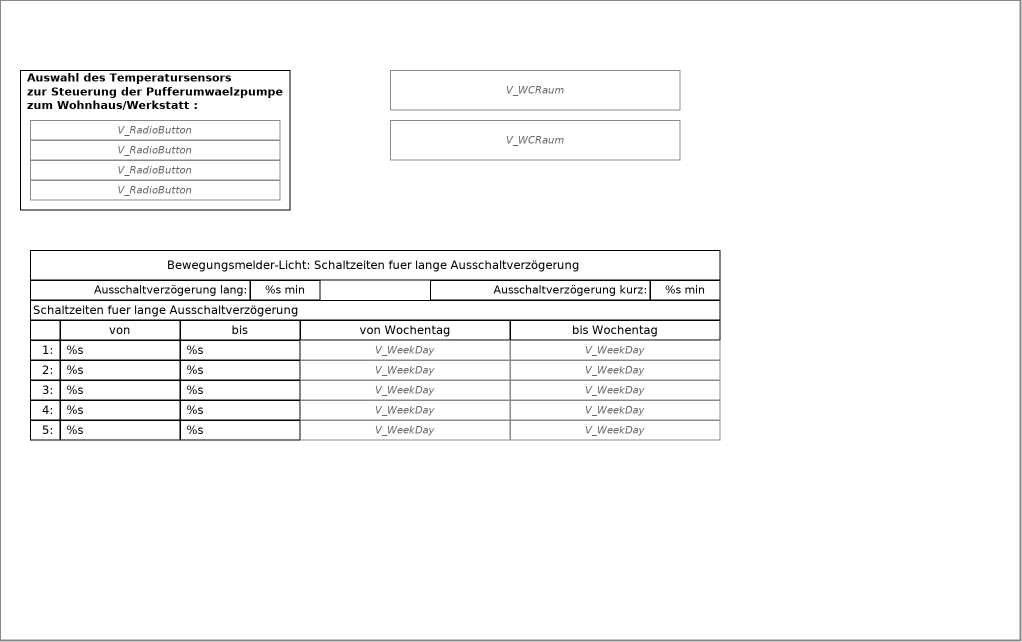
VISUALIZATION V_Einstellungen  // 1022x642
    Frame (0,-120 1020x760)
        shows V_Main_PC()
    Frame (390,120 290x40)
        shows V_WCRaum(IN_Title := 'WC Herren', IO_fbWCRaum := PLC_PRG.fbWCHerren)
    Frame (390,70 290x40)
        shows V_WCRaum(IN_Title := 'WC Damen', IO_fbWCRaum := PLC_PRG.fbWCDamen)
    Rectangle (20,70 270x140), "Auswahl des Temperatursensors zur Steuerung der Pufferumwaelzpumpe zum Wohnhaus/Werkstatt :", tooltip "Nach Abschalten des Bewegungsmelders läuft der Abluftventilator die hier eingestellte Zeit nach"
    Frame (30,120 250x20)
        shows V_RadioButton(IN_Title := '4000l-Puffer Brauchw.', IN_iValue := 4, IO_iVar := PLC_PRG.fbKompressorSteuerung.ViWRGTempSensorSelect)
    Frame (30,140 250x20)
        shows V_RadioButton(IN_Title := '4000l-Puffer oben', IN_iValue := 3, IO_iVar := PLC_PRG.fbKompressorSteuerung.ViWRGTempSensorSelect)
    Frame (30,160 250x20)
        shows V_RadioButton(IN_Title := '4000l-Puffer mitte', IN_iValue := 2, IO_iVar := PLC_PRG.fbKompressorSteuerung.ViWRGTempSensorSelect)
    Frame (30,180 250x20)
        shows V_RadioButton(IN_Title := '4000l-Puffer unten', IN_iValue := 1, IO_iVar := PLC_PRG.fbKompressorSteuerung.ViWRGTempSensorSelect)
    Rectangle (60,320 120x20), "von"
    Rectangle (60,340 120x20), "%s", text variable: VnvstSwitchTimesLichtBWMtofLang.todHeizEin[1]
        OnMouseDown: write the text variable via Edit
    Rectangle (30,340 30x20), "1:"
    Rectangle (30,250 690x30), "Bewegungsmelder-Licht: Schaltzeiten fuer lange Ausschaltverzögerung"
    Rectangle (30,360 30x20), "2:"
    Rectangle (30,380 30x20), "3:"
    Rectangle (30,400 30x20), "4:"
    Rectangle (30,420 30x20), "5:"
    Rectangle (180,320 120x20), "bis"
    Rectangle (30,320 30x20)
    Rectangle (180,340 120x20), "%s", text variable: VnvstSwitchTimesLichtBWMtofLang.todHeizAus[1]
        OnMouseDown: write the text variable via Edit
    Rectangle (300,320 210x20), "von Wochentag"
    Rectangle (510,320 210x20), "bis Wochentag"
    Rectangle (60,360 120x20), "%s", text variable: VnvstSwitchTimesLichtBWMtofLang.todHeizEin[2]
        OnMouseDown: write the text variable via Edit
    Rectangle (180,360 120x20), "%s", text variable: VnvstSwitchTimesLichtBWMtofLang.todHeizAus[2]
        OnMouseDown: write the text variable via Edit
    Rectangle (60,380 120x20), "%s", text variable: VnvstSwitchTimesLichtBWMtofLang.todHeizEin[3]
        OnMouseDown: write the text variable via Edit
    Rectangle (180,380 120x20), "%s", text variable: VnvstSwitchTimesLichtBWMtofLang.todHeizAus[3]
        OnMouseDown: write the text variable via Edit
    Rectangle (60,400 120x20), "%s", text variable: VnvstSwitchTimesLichtBWMtofLang.todHeizEin[4]
        OnMouseDown: write the text variable via Edit
    Rectangle (180,400 120x20), "%s", text variable: VnvstSwitchTimesLichtBWMtofLang.todHeizAus[4]
        OnMouseDown: write the text variable via Edit
    Rectangle (60,420 120x20), "%s", text variable: VnvstSwitchTimesLichtBWMtofLang.todHeizEin[5]
        OnMouseDown: write the text variable via Edit
    Rectangle (180,420 120x20), "%s", text variable: VnvstSwitchTimesLichtBWMtofLang.todHeizAus[5]
        OnMouseDown: write the text variable via Edit
    Rectangle (30,300 690x20), "Schaltzeiten fuer lange Ausschaltverzögerung"
    Rectangle (250,280 70x20), "%s min", tooltip "Nach Abschalten des Bewegungsmelders läuft der Abluftventilator die hier eingestellte Zeit nach", text variable: VnvdiLichtTofLang
        OnMouseClick: write the text variable via Default, min 3, max 600
    Rectangle (30,280 220x20), "Ausschaltverzögerung lang:", tooltip "Nach Abschalten des Bewegungsmelders läuft der Abluftventilator die hier eingestellte Zeit nach"
    Rectangle (430,280 220x20), "Ausschaltverzögerung kurz:", tooltip "Nach Abschalten des Bewegungsmelders läuft der Abluftventilator die hier eingestellte Zeit nach"
    Rectangle (650,280 70x20), "%s min", tooltip "Nach Abschalten des Bewegungsmelders läuft der Abluftventilator die hier eingestellte Zeit nach", text variable: VnvdiLichtTofKurz
        OnMouseClick: write the text variable via Default, min 0, max 30
    Frame (300,420 210x20)
        shows V_WeekDay(eWeekDay := VnvstSwitchTimesLichtBWMtofLang.eDayOfWeekStart[5])
    Frame (510,420 210x20)
        shows V_WeekDay(eWeekDay := VnvstSwitchTimesLichtBWMtofLang.eDayOfWeekEnd[5])
    Frame (300,340 210x20)
        shows V_WeekDay(eWeekDay := VnvstSwitchTimesLichtBWMtofLang.eDayOfWeekStart[1])
    Frame (510,340 210x20)
        shows V_WeekDay(eWeekDay := VnvstSwitchTimesLichtBWMtofLang.eDayOfWeekEnd[1])
    Frame (300,360 210x20)
        shows V_WeekDay(eWeekDay := VnvstSwitchTimesLichtBWMtofLang.eDayOfWeekStart[2])
    Frame (510,360 210x20)
        shows V_WeekDay(eWeekDay := VnvstSwitchTimesLichtBWMtofLang.eDayOfWeekEnd[2])
    Frame (300,380 210x20)
        shows V_WeekDay(eWeekDay := VnvstSwitchTimesLichtBWMtofLang.eDayOfWeekStart[3])
    Frame (510,380 210x20)
        shows V_WeekDay(eWeekDay := VnvstSwitchTimesLichtBWMtofLang.eDayOfWeekEnd[3])
    Frame (300,400 210x20)
        shows V_WeekDay(eWeekDay := VnvstSwitchTimesLichtBWMtofLang.eDayOfWeekStart[4])
    Frame (510,400 210x20)
        shows V_WeekDay(eWeekDay := VnvstSwitchTimesLichtBWMtofLang.eDayOfWeekEnd[4])
END_VISUALIZATION

(* stored: Version 1.1.0.1, ProductVersion 3.1.4018.9
   Visu V_Einstellungen: Id {abacb735-aa89-41cf-8c6d-1cf5f1d06192} *)
